(* Logix 5000 project; controller TEC_81 vendor 1 type 14 code 148 rev 36.11; software revision 36.00; part 5 of 5 *)
(* tags used below, declared in another part *)
   Lasers_OK : BOOL;   // Laser Scanner Close Loop Indicator
   Safety_Close_Loop_ok : BOOL;   // General Safety Indicator
   Safety_Mat_ok : BOOL;   // Safety Mat Close Loop Indicator
   TOF_STO_KinetixStorage1 : TIMER;
   EStops_OK : BOOL;   // E-Stop Close Loop Indicator
   Interlocks_Ok : BOOL;   // Interlocks Close Loop Indicator
   KUKA : TIMER;
   LigthCurtain_ok : BOOL;   // Light Curtains Close Loop Indicator
   Paro_Emergencia_Almacen_1 : BOOL;   // Stopping signal of Torc Off Almacen 1
   Paro_Emergencia_Almacen_2 : BOOL;   // Stopping signal of Torc Off Almacen 2
   TOF_STO_KinetixStorage2 : TIMER;
   TT : BOOL;
(* SafetyProgram, continued *)

ROUTINE SafetyCloseDoor   (* ladder *)
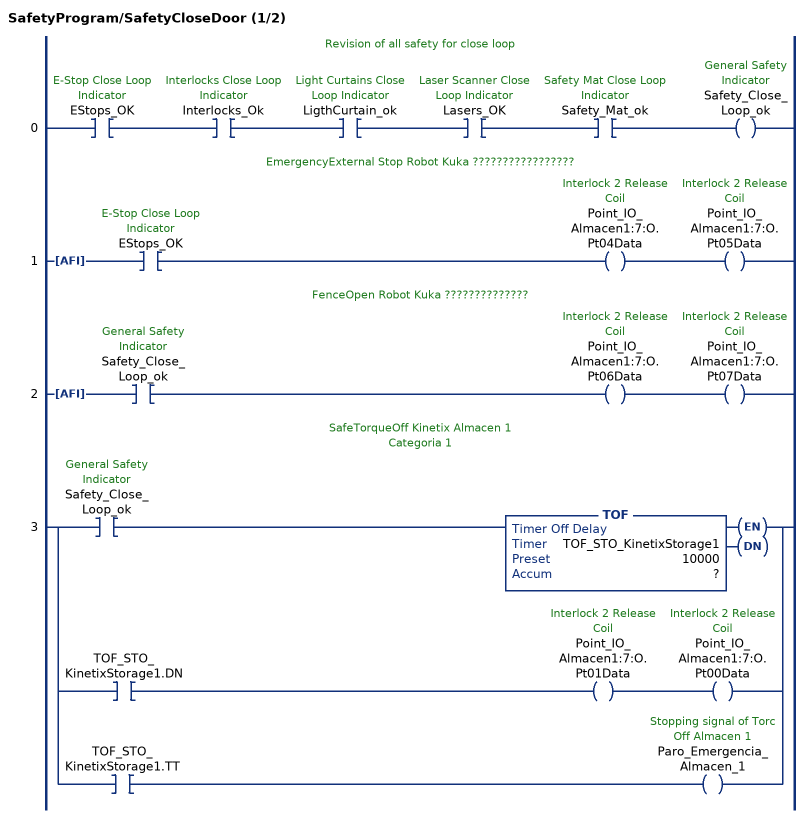
   // Revision of all safety for close loop
   0: XIC(EStops_OK)XIC(Interlocks_Ok)XIC(LigthCurtain_ok)XIC(Lasers_OK)XIC(Safety_Mat_ok)OTE(Safety_Close_Loop_ok);
   // EmergencyExternal Stop Robot Kuka ?????????????????
   1: AFI()XIC(EStops_OK)OTE(Point_IO_Almacen1:7:O.Pt04Data)OTE(Point_IO_Almacen1:7:O.Pt05Data);
   // FenceOpen Robot Kuka ??????????????
   2: AFI()XIC(Safety_Close_Loop_ok)OTE(Point_IO_Almacen1:7:O.Pt06Data)OTE(Point_IO_Almacen1:7:O.Pt07Data);
   // SafeTorqueOff Kinetix Almacen 1
   // Categoria 1
   3: [XIC(Safety_Close_Loop_ok) TOF(TOF_STO_KinetixStorage1,?,?) ,XIC(TOF_STO_KinetixStorage1.DN) OTE(Point_IO_Almacen1:7:O.Pt01Data) OTE(Point_IO_Almacen1:7:O.Pt00Data) ,XIC(TOF_STO_KinetixStorage1.TT) OTE(Paro_Emergencia_Almacen_1) ];
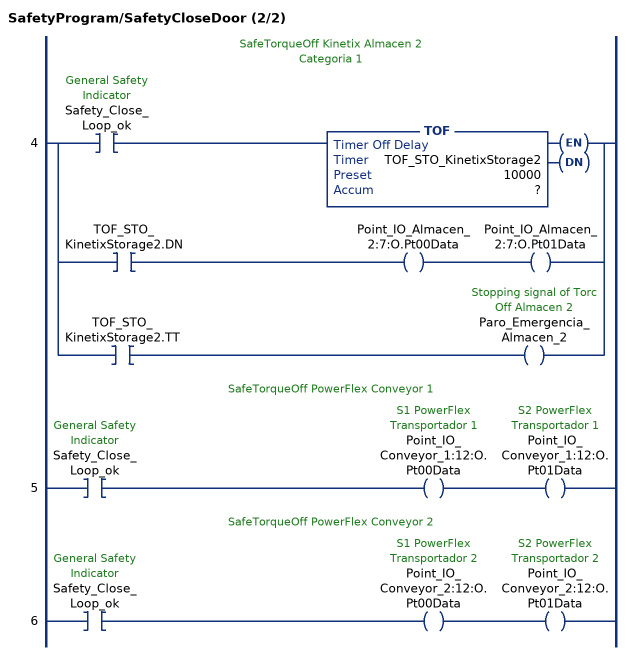
   // SafeTorqueOff Kinetix Almacen 2
   // Categoria 1
   4: [XIC(Safety_Close_Loop_ok) TOF(TOF_STO_KinetixStorage2,?,?) ,XIC(TOF_STO_KinetixStorage2.DN) OTE(Point_IO_Almacen_2:7:O.Pt00Data) OTE(Point_IO_Almacen_2:7:O.Pt01Data) ,XIC(TOF_STO_KinetixStorage2.TT) OTE(Paro_Emergencia_Almacen_2) ];
   // SafeTorqueOff PowerFlex Conveyor 1
   5: XIC(Safety_Close_Loop_ok)OTE(Point_IO_Conveyor_1:12:O.Pt00Data)OTE(Point_IO_Conveyor_1:12:O.Pt01Data);
   // SafeTorqueOff PowerFlex Conveyor 2
   6: XIC(Safety_Close_Loop_ok)OTE(Point_IO_Conveyor_2:12:O.Pt00Data)OTE(Point_IO_Conveyor_2:12:O.Pt01Data);
END_ROUTINE
END_PROGRAM
